FUNCTION_BLOCK PUBLIC ManualControl
VAR_INPUT
	Switch: BOOL;
END_VAR
VAR
	ManualControl: BOOL;
	TimeForInterlockDelay: TIME := T#0.05S;
	ManualMode: BOOL;
	MotorSelection_1: MotorSelection;
	SelectedMotor: WORD;
	temp: TIME;
	LowerLeftInterlock: TOF;
	LowerLeft: BOOL;
	LowerRightInterlock: TOF;
	LowerRight: BOOL;
END_VAR
VAR_OUTPUT
	Output: BOOL;
END_VAR
VAR // added by the converter: edge detectors and wires of the graphical bodies
    _w1, _w2, _w3, _w4, _w5, _w6, _w7, _w8, _w9, _w10, _w11 : BOOL;
    _rt1, _rt2, _rt3 : R_TRIG;
    _ft1, _ft2, _ft3 : F_TRIG;
END_VAR

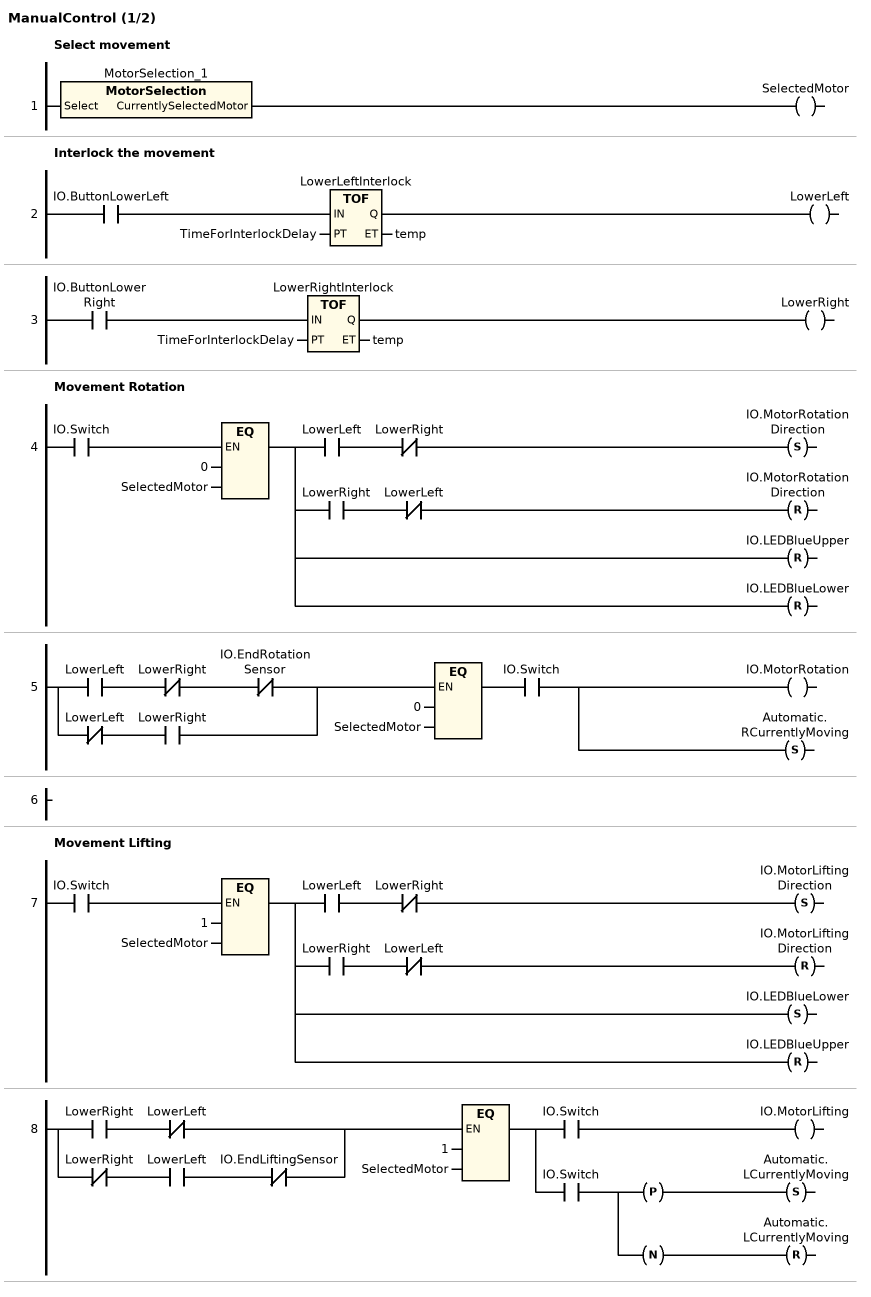
// NETWORK 1: Select movement
MotorSelection_1(Select := TRUE); // MotorSelection
SelectedMotor := MotorSelection_1.CurrentlySelectedMotor;

// NETWORK 2: Interlock the movement
LowerLeftInterlock(IN := IO.ButtonLowerLeft, PT := TimeForInterlockDelay, ET => temp); // TOF
LowerLeft := LowerLeftInterlock.Q;

// NETWORK 3
LowerRightInterlock(IN := IO.ButtonLowerRight, PT := TimeForInterlockDelay, ET => temp); // TOF
LowerRight := LowerRightInterlock.Q;

// NETWORK 4: Movement Rotation
_w1 := IO.Switch AND 0 = SelectedMotor;
IO.MotorRotationDirection S= _w1 AND LowerLeft AND NOT LowerRight;
IO.MotorRotationDirection R= _w1 AND LowerRight AND NOT LowerLeft;
IO.LEDBlueUpper R= _w1;
IO.LEDBlueLower R= _w1;

// NETWORK 5
_w2 := ((LowerLeft AND NOT LowerRight AND NOT IO.EndRotationSensor OR NOT LowerLeft AND LowerRight) AND 0 = SelectedMotor) AND IO.Switch;
IO.MotorRotation := _w2;
Automatic.RCurrentlyMoving S= _w2;

// NETWORK 6

// NETWORK 7: Movement Lifting
_w3 := IO.Switch AND 1 = SelectedMotor;
IO.MotorLiftingDirection S= _w3 AND LowerLeft AND NOT LowerRight;
IO.MotorLiftingDirection R= _w3 AND LowerRight AND NOT LowerLeft;
IO.LEDBlueLower S= _w3;
IO.LEDBlueUpper R= _w3;

// NETWORK 8
_w4 := (LowerRight AND NOT LowerLeft OR NOT LowerRight AND LowerLeft AND NOT IO.EndLiftingSensor) AND 1 = SelectedMotor;
IO.MotorLifting := _w4 AND IO.Switch;
_w5 := _w4 AND IO.Switch;
_rt1(CLK := _w5);
Automatic.LCurrentlyMoving S= _rt1.Q;
_ft1(CLK := _w5);
Automatic.LCurrentlyMoving R= _ft1.Q;

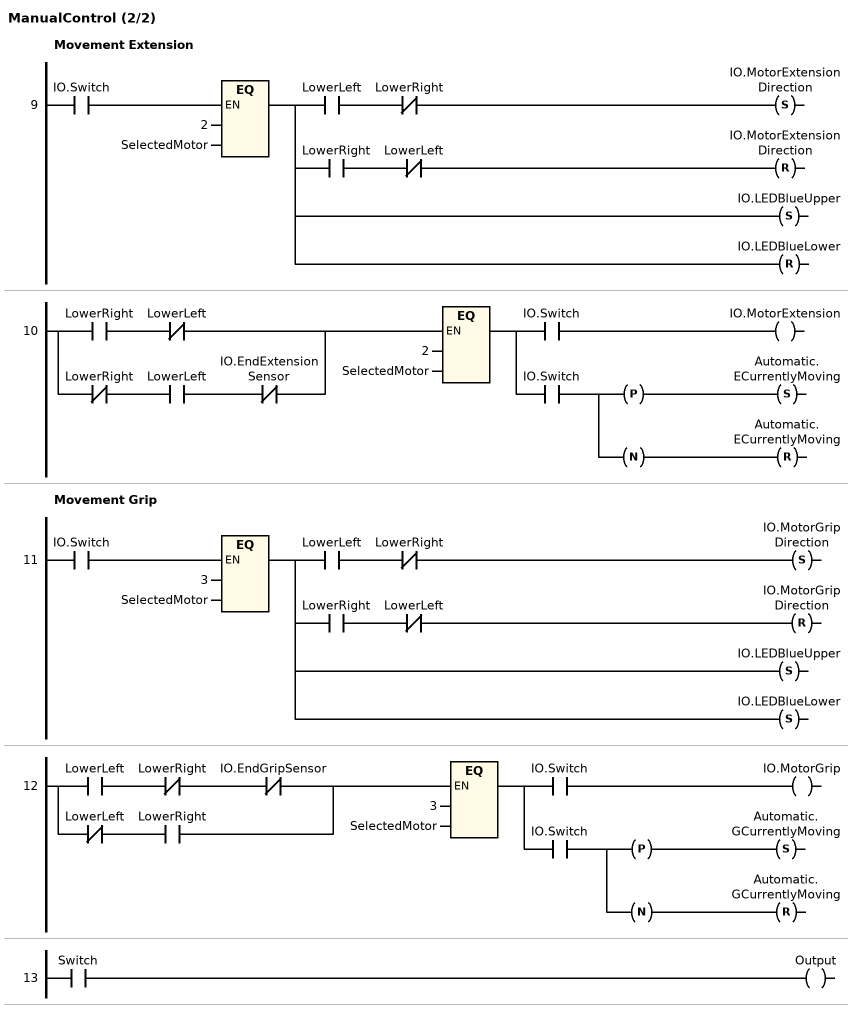
// NETWORK 9: Movement Extension
_w6 := IO.Switch AND 2 = SelectedMotor;
IO.MotorExtensionDirection S= _w6 AND LowerLeft AND NOT LowerRight;
IO.MotorExtensionDirection R= _w6 AND LowerRight AND NOT LowerLeft;
IO.LEDBlueUpper S= _w6;
IO.LEDBlueLower R= _w6;

// NETWORK 10
_w7 := (LowerRight AND NOT LowerLeft OR NOT LowerRight AND LowerLeft AND NOT IO.EndExtensionSensor) AND 2 = SelectedMotor;
IO.MotorExtension := _w7 AND IO.Switch;
_w8 := _w7 AND IO.Switch;
_rt2(CLK := _w8);
Automatic.ECurrentlyMoving S= _rt2.Q;
_ft2(CLK := _w8);
Automatic.ECurrentlyMoving R= _ft2.Q;

// NETWORK 11: Movement Grip
_w9 := IO.Switch AND 3 = SelectedMotor;
IO.MotorGripDirection S= _w9 AND LowerLeft AND NOT LowerRight;
IO.MotorGripDirection R= _w9 AND LowerRight AND NOT LowerLeft;
IO.LEDBlueUpper S= _w9;
IO.LEDBlueLower S= _w9;

// NETWORK 12
_w10 := (LowerLeft AND NOT LowerRight AND NOT IO.EndGripSensor OR NOT LowerLeft AND LowerRight) AND 3 = SelectedMotor;
IO.MotorGrip := _w10 AND IO.Switch;
_w11 := _w10 AND IO.Switch;
_rt3(CLK := _w11);
Automatic.GCurrentlyMoving S= _rt3.Q;
_ft3(CLK := _w11);
Automatic.GCurrentlyMoving R= _ft3.Q;

// NETWORK 13
Output := Switch;

END_FUNCTION_BLOCK

(* stored: Version 1.1.0.1, ProductVersion 3.1.4024.13
   POU ManualControl: Id {0dc011e3-56d5-4b91-a8d5-8c19aa1fc8c8}, SpecialFunc None *)
